{attribute 'qualified_only'}
VAR_GLOBAL
    // Kompanzasyon grupları konfigürasyonu
    astCompensationGroups : ARRAY[0..GVL_CompensationGroup.MAX_COMPENSATION_GROUPS-1] OF ST_CompensationGroup;  // Tüm grupların kondansatör bilgileri
    nConfiguredGroups : INT;                                                                                    // Toplam konfigüre edilmiş grup sayısı
    
    // Grup aktif durumları
    abGroupActive : ARRAY[0..GVL_CompensationGroup.MAX_COMPENSATION_GROUPS-1] OF BOOL;                         // Her grubun aktif/pasif durumu

    // Ana kesici HMI bilgileri
    stMainDisconnectorHMI : ST_DisconnectorHMI;                                                               // Ana kesici durum ve kontrol bilgileri	
	
	// 12CB1 kesici HMI bilgileri
	st12CB1HMI : ST_DisconnectorHMI;		// 12CB1 kesici durum ve kontrol bilgileri		
	
	// 14CB1 kesici HMI bilgileri
	st14CB1HMI : ST_DisconnectorHMI;		// 14CB1 kesici durum ve kontrol bilgileri	
	
	// 16CB1 kesici HMI bilgileri
	st16CB1HMI : ST_DisconnectorHMI;		// 16CB1 kesici durum ve kontrol bilgileri
	
	// 18CB1 kesici HMI bilgileri
	st18CB1HMI : ST_DisconnectorHMI;		// 18CB1 kesici durum ve kontrol bilgileri
	
	// 20CB1 kesici HMI bilgileri
	st20CB1HMI : ST_DisconnectorHMI;		// 20CB1 kesici durum ve kontrol bilgileri
	
	// 22CB1 kesici HMI bilgileri
	st22CB1HMI : ST_DisconnectorHMI;		// 22CB1 kesici durum ve kontrol bilgileri
	
	// 24CB1 kesici HMI bilgileri
	st24CB1HMI : ST_DisconnectorHMI;		// 24CB1 kesici durum ve kontrol bilgileri
	
	// 26CB1 kesici HMI bilgileri
	st26CB1HMI : ST_DisconnectorHMI;		// 26CB1 kesici durum ve kontrol bilgileri
	
	// 28CB1 kesici HMI bilgileri
	st28CB1HMI : ST_DisconnectorHMI;		// 28CB1 kesici durum ve kontrol bilgileri
	
	// 30CB1 kesici HMI bilgileri
	st30CB1HMI : ST_DisconnectorHMI;		// 30CB1 kesici durum ve kontrol bilgileri
	
	// 32CB1 kesici HMI bilgileri
	st32CB1HMI : ST_DisconnectorHMI;		// 32CB1 kesici durum ve kontrol bilgileri
	
	// 34CB1 kesici HMI bilgileri
	st34CB1HMI : ST_DisconnectorHMI;		// 34CB1 kesici durum ve kontrol bilgileri
	
	// 36CB1 kesici HMI bilgileri
	st36CB1HMI : ST_DisconnectorHMI;		// 36CB1 kesici durum ve kontrol bilgileri
	
	// 38CB1 kesici HMI bilgileri
	st38CB1HMI : ST_DisconnectorHMI;		// 38CB1 kesici durum ve kontrol bilgileri
	
	// 40CB1 kesici HMI bilgileri
	st40CB1HMI : ST_DisconnectorHMI;		// 40CB1 kesici durum ve kontrol bilgileri
	
	// 42CB1 kesici HMI bilgileri
	st42CB1HMI : ST_DisconnectorHMI;		// 42CB1 kesici durum ve kontrol bilgileri
	
	// 44CB1 kesici HMI bilgileri
	st44CB1HMI : ST_DisconnectorHMI;		// 44CB1 kesici durum ve kontrol bilgileri
	
	// 46CB1 kesici HMI bilgileri
	st46CB1HMI : ST_DisconnectorHMI;		// 46CB1 kesici durum ve kontrol bilgileri
	
	// 48CB1 kesici HMI bilgileri
	st48CB1HMI : ST_DisconnectorHMI;		// 48CB1 kesici durum ve kontrol bilgileri
	
	// 50CB1 kesici HMI bilgileri
	st50CB1HMI : ST_DisconnectorHMI;		// 50CB1 kesici durum ve kontrol bilgileri
	
	// 52CB1 kesici HMI bilgileri
	st52CB1HMI : ST_DisconnectorHMI;		// 52CB1 kesici durum ve kontrol bilgileri
	
	// 54CB1 kesici HMI bilgileri
	st54CB1HMI : ST_DisconnectorHMI;		// 54CB1 kesici durum ve kontrol bilgileri
	
	// 56CB1 kesici HMI bilgileri
	st56CB1HMI : ST_DisconnectorHMI;		// 56CB1 kesici durum ve kontrol bilgileri
	
END_VAR

(* stored: Version 1.1.0.1, ProductVersion 3.1.4024.15
   GVL GVL_HVCP3: Id {79487589-2562-43b6-9dd8-3f72c84a3823} *)
